// TIA Portal project "OPC_UA_STEP7_CODE_V12" (V14)

(* hardware
DEVICE "SIMATIC 300"  S7-300 station
   slot 0: "UR"  Rail  6ES7 390-1***0-0AA0
   slot 2: "CPU 315-2 PN/DP"  CPU 315-2 PN/DP  6ES7 315-2EH14-0AB0  V3.2
      slot 2: "PROFINET interface_1"  PN-IO
         slot 1: "Port_1"  Port
         slot 2: "Port_2"  Port
   slot 4: "CP 343-1 Advanced-IT_1"  CP 343-1 ADVANCED-IT  6GK7 343-1GX31-0XE0  V3.0
   slot 5: "DI 16/DO 16x24VDC/0.5A"  DI16/DO16 x 24V / 0.5A  6ES7 323-1BL00-0AA0
DEVICE "SIMATIC 400"  S7-400 station
   slot 0: "UR2"  UR2ALU-H  6ES7 400-1JA01-0AA0
   slot 1: "PS 407 10A"  PS 407 10A  6ES7 407-0KA02-0AA0
   slot 3: "CPU 416-3 DP"  CPU 416-3DP  6ES7 416-3XR05-0AB0  V5.1
      slot 1: "DP"  X2
      slot 2: "MPI/DP"  X1
   slot 5: "CP 443-1 Advanced"  CP 443-1 Advanced-IT  6GK7 443-1GX20-0XE0  V2.0
   slot 6: "SM 423 SIM"  DI/DO SIMULATOR  6ES7 423 DI/DO-SIMULATOR
DEVICE "SIMATIC PC Station"  SIMATIC PC station
   slot 0: "PC"  Rail  SIMATIC PC-Station  V1.0
      slot 125: "Stationmanager"  Station_Manager  V6.0.4
   slot 1: "OPC Server"  OPC Server  OPC Server  V14.0.0
   slot 2: "IE General"  IE General  IE_CP  V8.2.0
DEVICE "S71500/ET200MP station_1"  S7-1500 station
   slot 0: "Rail_0"  Rack  6ES7 590-1***0-0AA0
   slot 1: "CPU 1516F-3 PN/DP"  CPU 1516F-3 PN/DP  6ES7 516-3FN00-0AB0  V1.8
      slot 3: "CPU display_1"  6ES7591-1BA00-0AA0
*)

// ===== PLC "CPU 315-2 PN/DP"  CPU 315-2 PN/DP =====

VAR_GLOBAL   // PLC tag table "Default tag table"
   "Tag_1" AT %M100.1 : Bool;
   "Tag_2" AT %M10.6 : Bool;
   "Tag_3" AT %MW302 : Int;
   "Tag_4" AT %MW300 : Int;
   "Tag_5" AT %T1 : Timer;
   "Tag_6" AT %M100.0 : Bool;
END_VAR

VAR_GLOBAL   // PLC tag table "STEP7 classic symbols"
   "CountUP" AT %MB10 : Byte;
END_VAR

DATA_BLOCK "SimulationConfiguration"   // DB10
{ S7_Optimized_Access := 'FALSE' }
VERSION : 0.1
   VAR
      SimulationSpeed : Byte := B#16#10;
      DynamicCharacter : Byte := B#16#20;
      StartASCII : Byte := B#16#20;
      EndASCII : Byte := B#16#7F;
      CurrentStringLength : Byte := B#16#A;
      MaxStringLength : Byte := B#16#A;
      SendDataCountUp : Byte;
      SendDataLength : DWord := DW#16#1000;
   END_VAR
BEGIN
END_DATA_BLOCK

DATA_BLOCK "StaticDataTypes"   // DB50
{ S7_Optimized_Access := 'FALSE' }
VERSION : 0.1
   VAR
      My_Bool : Bool := TRUE;   // Temporary placeholder variable
      My_Integer : Int := -32767;
      My_Byte : Byte := B#16#FF;
      My_Word : Word := W#16#FFFF;
      My_DWord : DWord := DW#16#FFFFFFFF;
      My_DInteger : DInt := L#-2147483647;
      My_Real4 : Real := 1.23456e+0;
      My_Char : Char := 'a';
      My_String10 : String[10] := 'HelloWorld';
      My_DateAndTime : Date_And_Time := DT#10-12-31-12:59:59.123;
   END_VAR
BEGIN
END_DATA_BLOCK

DATA_BLOCK "DynamicDataTypes"   // DB51
{ S7_Optimized_Access := 'FALSE' }
VERSION : 0.1
   VAR
      My_Bool : Bool;   // Temporary placeholder variable
      My_Integer : Int;
      My_Byte : Byte;
      My_Word : Word;
      My_DWord : DWord;
      My_DInteger : DInt;
      My_Real4 : Real;
      My_Char : Char;
      My_String10 : String[10];
      My_DateAndTime : Date_And_Time;
   END_VAR
BEGIN
END_DATA_BLOCK

DATA_BLOCK "InstanceDataBSEND-BRCV"   // DB100
{ S7_Optimized_Access := 'FALSE' }
VERSION : 0.0
// stored: InstanceOfName InvokeBSENDandBRCV
"InvokeBSENDandBRCV"
BEGIN
   BSEND.SD_1 := P#P  0.0 VOID 0;
   BRCV.RD_1 := P#P  0.0 VOID 0;
END_DATA_BLOCK

DATA_BLOCK "SendData"   // DB112
{ S7_Optimized_Access := 'FALSE' }
VERSION : 0.1
   VAR
      SendData : Array[0..4096] of Byte;
   END_VAR
BEGIN
END_DATA_BLOCK

DATA_BLOCK "RcvData"   // DB113
{ S7_Optimized_Access := 'FALSE' }
VERSION : 0.1
   VAR
      RcvData : Array[0..4096] of Byte;
   END_VAR
BEGIN
END_DATA_BLOCK

FUNCTION_BLOCK "InvokeBSENDandBRCV"   // FB100, STL
{ S7_Optimized_Access := 'FALSE' }
VERSION : 0.1
   VAR_INPUT
      INIT_COM : Bool;
   END_VAR
   VAR
      PLC1_COM : Struct
         BSEND_REQ : Bool;
         BSEND_BUSY : Bool;
         BSEND_DONE : Bool;
         BSEND_ERROR : Bool;
         BSEND_COM_START : Bool;   // Pos flank
         BRCV_EN_R : Bool;
         BRCV_BUSY : Bool;
         BRCV_NDR : Bool;
         BRCV_ERROR : Bool;
         BRCV_COM_START : Bool;
         ID : Word;
         BSEND_STATUS : Word;
         BSEND_STAT_SAVE : Word;
         BRCV_STATUS : Word;
         BRCV_STAT_SAVE : Word;
         BSEND_LEN : Word;
         BRCV_LEN : Word;
      END_STRUCT;
      BSEND : BSEND;
      BRCV : BRCV;
   END_VAR
BEGIN

REGION Network 1: Clear BSEND request to start initial communication
         A     #INIT_COM;
         R     #PLC1_COM.BSEND_REQ;
END_REGION

REGION Network 2
   // define the LEN
         A     #INIT_COM;
         JNB   _001;
         L     "SimulationConfiguration".SendDataLength;
         T     #PLC1_COM.BSEND_LEN;
   _001: NOP   0;
END_REGION

REGION Network 3: Invoke BSEND function
         A     #PLC1_COM.BSEND_REQ;
         =     <??.?>;
         BLD   103;
         A     "Tag_1";
         JNB   _002;
         CALL  #BSEND
         ( REQ    := <??.?>,
           R      := ,
           ID     := 16#0001,
           R_ID   := 16#0000_0002,
           DONE   := #PLC1_COM.BSEND_DONE,
           ERROR  := #PLC1_COM.BSEND_ERROR,
           STATUS := #PLC1_COM.BSEND_STATUS,
           SD_1   := P#DB112.DBX0.0 BYTE 4096,
           LEN    := #PLC1_COM.BSEND_LEN
         );
   _002: NOP   0;
END_REGION

REGION Network 4
   // Start BSEND function with the rising edge of the clock marker if the BSEND 
   // function is not busy
   // The REQ input parameter of the BSEND function is triggered with a rising edge 
   // as 
   // long as the BSEND function is not completed!
         AN    "Tag_2";
         S     #PLC1_COM.BSEND_REQ;
         A(;
         O     #PLC1_COM.BSEND_ERROR;
         O     #PLC1_COM.BSEND_DONE;
         );
         R     #PLC1_COM.BSEND_REQ;
         NOP   0;
END_REGION

REGION Network 5: Evaluate STATUS information of the BSEND function
   // If ERROR occured then save STATUS!
         A     #PLC1_COM.BSEND_ERROR;
         JNB   _003;
         L     #PLC1_COM.BSEND_STATUS;
         T     #PLC1_COM.BSEND_STAT_SAVE;
   _003: NOP   0;
END_REGION

REGION Network 6: Invoke BRCV function
         A     "Tag_1";
         =     <??.?>;
         BLD   103;
         A     "Tag_1";
         JNB   _004;
         CALL  #BRCV
         ( EN_R   := <??.?>,
           ID     := 16#0001,
           R_ID   := 16#0000_0001,
           NDR    := #PLC1_COM.BRCV_NDR,
           ERROR  := #PLC1_COM.BRCV_ERROR,
           STATUS := #PLC1_COM.BRCV_STATUS,
           RD_1   := P#DB113.DBX0.0 BYTE 4096,
           LEN    := #PLC1_COM.BRCV_LEN
         );
   _004: NOP   0;
END_REGION

REGION Network 7: Evaluate STATUS information of the BRCV function
   // If ERROR occured then save STATUS!
         A     #PLC1_COM.BRCV_ERROR;
         JNB   _005;
         L     #PLC1_COM.BRCV_STATUS;
         T     #PLC1_COM.BRCV_STAT_SAVE;
   _005: NOP   0;
END_REGION

REGION Network 8: Enable output ENO
         A     "Tag_1";
         SAVE;
END_REGION
END_FUNCTION_BLOCK

FUNCTION "ChangeDateAndTime" : Void   // FC10, STL
{ S7_Optimized_Access := 'FALSE' }
VERSION : 0.1
BEGIN

REGION Network 1
   // Dynamic Date and Time
   //// year
         L     99;
         L     %DB51.DBB34;
         BTI;
         +     1;
         <I;
         JCN   no1;
         L     0;
   no1:  ITB;
         T     %DB51.DBB34;
   //// month
         L     12;
         L     %DB51.DBB35;
         BTI;
         +     1;
         <I;
         JCN   no2;
         L     1;
   no2:  ITB;
         T     %DB51.DBB35;
   //// day
         L     31;
         L     %DB51.DBB36;
         BTI;
         +     1;
         <I;
         JCN   no3;
         L     1;
   no3:  ITB;
         T     %DB51.DBB36;
   //// hour
         L     23;
         L     %DB51.DBB37;
         BTI;
         +     1;
         <I;
         JCN   no4;
         L     0;
   no4:  ITB;
         T     %DB51.DBB37;
   //// minute
         L     59;
         L     %DB51.DBB38;
         BTI;
         +     1;
         <I;
         JCN   no5;
         L     0;
   no5:  ITB;
         T     %DB51.DBB38;
   //// second
         L     59;
         L     %DB51.DBB39;
         BTI;
         +     1;
         <I;
         JCN   no6;
         L     0;
   no6:  ITB;
         T     %DB51.DBB39;
   //// millisecond left part
         L     99;
         L     %DB51.DBB40;
         BTI;
         +     1;
         <I;
         JCN   no7;
         L     0;
   no7:  ITB;
         T     %DB51.DBB40;
   //// millisecond right part
         L     90;
         L     %DB51.DBB41;
         BTI;
         +     10;
         <I;
         JCN   no8;
         L     0;
   no8:  ITB;
         T     %DB51.DBB41;
END_REGION
END_FUNCTION

FUNCTION "ChangeSimpleTypes" : Void   // FC11, STL
{ S7_Optimized_Access := 'FALSE' }
VERSION : 0.1
BEGIN

REGION Network 1: Temporary placeholder variable
   // togle the boolean
         AN    "DynamicDataTypes".My_Bool;
         =     "DynamicDataTypes".My_Bool;
   // increment the byte
         L     "DynamicDataTypes".My_Byte;
         +     1;
         T     "DynamicDataTypes".My_Byte;
   // increment the signed byte
         L     "DynamicDataTypes".My_Char;
         +     1;
         T     "DynamicDataTypes".My_Char;
   // count up by 10
         L     "DynamicDataTypes".My_Word;
         +     10;
         T     "DynamicDataTypes".My_Word;
   // count up by 100
         L     "DynamicDataTypes".My_DWord;
         +     100;
         T     "DynamicDataTypes".My_DWord;
   // count up by 10
         L     "DynamicDataTypes".My_Integer;
         +     10;
         T     "DynamicDataTypes".My_Integer;
   // count up by 100
         L     "DynamicDataTypes".My_DInteger;
         +     100;
         T     "DynamicDataTypes".My_DInteger;
   // count up by 0.1
         L     "DynamicDataTypes".My_Real4;
         L     0.01;
         +R;
         T     "DynamicDataTypes".My_Real4;
END_REGION
END_FUNCTION

FUNCTION "ChangeString" : Void   // FC13, STL
{ S7_Optimized_Access := 'FALSE' }
VERSION : 0.1
BEGIN

REGION Network 1
   // change the content and the length of the string
   // Increment length of dynamic string 10
         L     "SimulationConfiguration".CurrentStringLength;
         L     "SimulationConfiguration".MaxStringLength;
         >=I;
         JC    rst1;

         L     "SimulationConfiguration".CurrentStringLength;
         +     1;
         T     "SimulationConfiguration".CurrentStringLength;
         T     %DB51.DBB23;  //used length of string
         JU    go1;

   rst1: L     1;
         T     "SimulationConfiguration".CurrentStringLength;
         T     %DB51.DBB23;


   // Set new StringChar
   go1:  L     "SimulationConfiguration".DynamicCharacter;
         L     "SimulationConfiguration".EndASCII;  // this is the last letter (ASCII) to use
         >=I;
         JC    rst2;

         L     "SimulationConfiguration".DynamicCharacter;
         +     1;
         T     "SimulationConfiguration".DynamicCharacter;
         JU    go2;

   rst2: L     "SimulationConfiguration".StartASCII;  // this is the first letter (ASCII) to use (32)
         T     "SimulationConfiguration".DynamicCharacter;

   go2:  CALL  FILL
         ( BVAL    := "SimulationConfiguration".DynamicCharacter,
           RET_VAL := "Tag_3",
           BLK     := P#DB51.DBX24.0 BYTE 10
         );
END_REGION
END_FUNCTION

FUNCTION "ChangeSendData" : Void   // FC14, STL
{ S7_Optimized_Access := 'FALSE' }
VERSION : 0.1
BEGIN

REGION Network 1

         L     "SimulationConfiguration".SendDataCountUp;
         L     1;
         +I;
         T     "SimulationConfiguration".SendDataCountUp;
   // take the byte and fill the send buffer
         CALL  FILL
         ( BVAL    := "SimulationConfiguration".SendDataCountUp,
           RET_VAL := "Tag_4",
           BLK     := P#DB112.DBX0.0 BYTE 4096
         );
         NOP   0;
END_REGION
END_FUNCTION

ORGANIZATION_BLOCK "OB1"   // OB1, STL
{ S7_Optimized_Access := 'FALSE' }
VERSION : 0.1
   VAR_TEMP
      TEMP0 : Byte;
      TEMP1 : Byte;
      TEMP2 : Byte;
      TEMP3 : Byte;
      TEMP4 : Byte;
      TEMP5 : Byte;
      TEMP6 : Int;
      TEMP7 : Int;
      TEMP8 : Int;
      TEMP9 : Date_And_Time;
   END_VAR
BEGIN

REGION Network 1: Get a trigger, speed depends on DB10 byte 0
   // check if timer is expired
         AN    "Tag_5";
   // start timer with value global speed variable
         L     "SimulationConfiguration".SimulationSpeed;
         ITB;
         SF    "Tag_5";
         JCN   END;

   // change the values

         CALL  "ChangeDateAndTime";

         CALL  "ChangeSimpleTypes";

         CALL  "ChangeString";

         CALL  "ChangeSendData";

   END:  NOP   0;
END_REGION

REGION Network 2: Activate communication with BSEND/BRCV function
         A     "Tag_6";
         =     <??.?>;
         BLD   103;
         A     "Tag_1";
         JNB   _001;
         CALL  "InvokeBSENDandBRCV", "InstanceDataBSEND-BRCV"
         ( INIT_COM := <??.?>
         );

   _001: A     BR;
         R     "Tag_6";
END_REGION
END_ORGANIZATION_BLOCK

ORGANIZATION_BLOCK "OB100"   // OB100, STL
TITLE = "Complete Restart"
{ S7_Optimized_Access := 'FALSE' }
VERSION : 0.1
   VAR_TEMP
      OB100_EV_CLASS : Byte;   // 16#13, Event class 1, Entering event state, Event logged in diagnostic buffer
      OB100_STRTUP : Byte;   // 16#81/82/83/84 Method of startup
      OB100_PRIORITY : Byte;   // Priority of OB Execution
      OB100_OB_NUMBR : Byte;   // 100 (Organization block 100, OB100)
      OB100_RESERVED_1 : Byte;   // Reserved for system
      OB100_RESERVED_2 : Byte;   // Reserved for system
      OB100_STOP : Word;   // Event that caused CPU to stop (16#4xxx)
      OB100_STRT_INFO : DWord;   // Information on how system started
      OB100_DATE_TIME : Date_And_Time;   // Date and time OB100 started
   END_VAR
BEGIN

REGION Network 1: Enable communication function blocks

         AN    "Tag_6";
         S     "Tag_6";
END_REGION

REGION Network 2: Force restart of communication block
         AN    "Tag_1";
         S     "Tag_1";
END_REGION
END_ORGANIZATION_BLOCK

// ===== PLC "CPU 416-3 DP"  CPU 416-3DP =====

VAR_GLOBAL   // PLC tag table "Default tag table"
   "Tag_1" AT %M100.1 : Bool;
   "Tag_2" AT %M10.6 : Bool;
   "Tag_3" AT %MW302 : Int;
   "Tag_4" AT %MW300 : Int;
   "Tag_5" AT %T1 : Timer;
   "Tag_6" AT %M100.0 : Bool;
END_VAR

VAR_GLOBAL   // PLC tag table "STEP7 classic symbols"
   "CountUP" AT %MB10 : Byte;
END_VAR

DATA_BLOCK "SimulationConfiguration"   // DB10
{ S7_Optimized_Access := 'FALSE' }
VERSION : 0.1
   VAR
      SimulationSpeed : Byte := B#16#10;
      DynamicCharacter : Byte := B#16#20;
      StartASCII : Byte := B#16#20;
      EndASCII : Byte := B#16#7F;
      CurrentStringLength : Byte := B#16#A;
      MaxStringLength : Byte := B#16#A;
      SendDataCountUp : Byte;
      SendDataLength : DWord := DW#16#1000;
   END_VAR
BEGIN
END_DATA_BLOCK

DATA_BLOCK "StaticDataTypes"   // DB50
{ S7_Optimized_Access := 'FALSE' }
VERSION : 0.1
   VAR
      My_Bool : Bool := TRUE;   // Temporary placeholder variable
      My_Integer : Int := -32767;
      My_Byte : Byte := B#16#FF;
      My_Word : Word := W#16#FFFF;
      My_DWord : DWord := DW#16#FFFFFFFF;
      My_DInteger : DInt := L#-2147483647;
      My_Real4 : Real := 1.23456e+0;
      My_Char : Char := 'a';
      My_String10 : String[10] := 'HelloWorld';
      My_DateAndTime : Date_And_Time := DT#10-12-31-12:59:59.123;
   END_VAR
BEGIN
END_DATA_BLOCK

DATA_BLOCK "DynamicDataTypes"   // DB51
{ S7_Optimized_Access := 'FALSE' }
VERSION : 0.1
   VAR
      My_Bool : Bool;   // Temporary placeholder variable
      My_Integer : Int;
      My_Byte : Byte;
      My_Word : Word;
      My_DWord : DWord;
      My_DInteger : DInt;
      My_Real4 : Real;
      My_Char : Char;
      My_String10 : String[10];
      My_DateAndTime : Date_And_Time;
   END_VAR
BEGIN
END_DATA_BLOCK

DATA_BLOCK "InstanceDataBSEND-BRCV"   // DB100
{ S7_Optimized_Access := 'FALSE' }
VERSION : 0.0
// stored: InstanceOfName InvokeBSENDandBRCV
"InvokeBSENDandBRCV"
BEGIN
END_DATA_BLOCK

DATA_BLOCK "SendData"   // DB112
{ S7_Optimized_Access := 'FALSE' }
VERSION : 0.1
   VAR
      SendData : Array[0..4096] of Byte;
   END_VAR
BEGIN
END_DATA_BLOCK

DATA_BLOCK "RcvData"   // DB113
{ S7_Optimized_Access := 'FALSE' }
VERSION : 0.1
   VAR
      RcvData : Array[0..4096] of Byte;
   END_VAR
BEGIN
END_DATA_BLOCK

FUNCTION_BLOCK "InvokeBSENDandBRCV"   // FB100, STL
{ S7_Optimized_Access := 'FALSE' }
VERSION : 0.1
   VAR_INPUT
      INIT_COM : Bool;
   END_VAR
   VAR
      PLC1_COM : Struct
         BSEND_REQ : Bool;
         BSEND_BUSY : Bool;
         BSEND_DONE : Bool;
         BSEND_ERROR : Bool;
         BSEND_COM_START : Bool;   // Pos flank
         BRCV_EN_R : Bool;
         BRCV_BUSY : Bool;
         BRCV_NDR : Bool;
         BRCV_ERROR : Bool;
         BRCV_COM_START : Bool;
         ID : Word;
         BSEND_STATUS : Word;
         BSEND_STAT_SAVE : Word;
         BRCV_STATUS : Word;
         BRCV_STAT_SAVE : Word;
         BSEND_LEN : Word;
         BRCV_LEN : Word;
      END_STRUCT;
   END_VAR
BEGIN

REGION Network 1: Clear BSEND request to start initial communication
         A     #INIT_COM;
         R     #PLC1_COM.BSEND_REQ;
END_REGION

REGION Network 2
   // define the LEN
         A     #INIT_COM;
         JNB   _001;
         L     "SimulationConfiguration".SendDataLength;
         T     #PLC1_COM.BSEND_LEN;
   _001: NOP   0;
END_REGION

REGION Network 3: Invoke BSEND function
         A     #PLC1_COM.BSEND_REQ;
         =     <??.?>;
         BLD   103;
         A     "Tag_1";
         JNB   _002;
         CALL  BSEND, "DB12"
         ( REQ    := <??.?>,
           R      := ,
           ID     := 16#0001,
           R_ID   := 16#0000_0001,
           DONE   := #PLC1_COM.BSEND_DONE,
           ERROR  := #PLC1_COM.BSEND_ERROR,
           STATUS := #PLC1_COM.BSEND_STATUS,
           SD_1   := P#DB112.DBX0.0 BYTE 4096,
           LEN    := #PLC1_COM.BSEND_LEN
         );
   _002: NOP   0;
END_REGION

REGION Network 4
   // Start BSEND function with the rising edge of the clock marker if the BSEND 
   // function is not busy
   // The REQ input parameter of the BSEND function is triggered with a rising edge 
   // as 
   // long as the BSEND function is not completed!
         AN    "Tag_2";
         S     #PLC1_COM.BSEND_REQ;
         A(;
         O     #PLC1_COM.BSEND_ERROR;
         O     #PLC1_COM.BSEND_DONE;
         );
         R     #PLC1_COM.BSEND_REQ;
         NOP   0;
END_REGION

REGION Network 5: Evaluate STATUS information of the BSEND function
   // If ERROR occured then save STATUS!
         A     #PLC1_COM.BSEND_ERROR;
         JNB   _003;
         L     #PLC1_COM.BSEND_STATUS;
         T     #PLC1_COM.BSEND_STAT_SAVE;
   _003: NOP   0;
END_REGION

REGION Network 6: Invoke BRCV function
         A     "Tag_1";
         =     <??.?>;
         BLD   103;
         A     "Tag_1";
         JNB   _004;
         CALL  BRCV, "DB13"
         ( EN_R   := <??.?>,
           ID     := 16#0001,
           R_ID   := 16#0000_0001,
           NDR    := #PLC1_COM.BRCV_NDR,
           ERROR  := #PLC1_COM.BRCV_ERROR,
           STATUS := #PLC1_COM.BRCV_STATUS,
           RD_1   := P#DB113.DBX0.0 BYTE 4096,
           LEN    := #PLC1_COM.BRCV_LEN
         );
   _004: NOP   0;
END_REGION

REGION Network 7: Evaluate STATUS information of the BRCV function
   // If ERROR occured then save STATUS!
         A     #PLC1_COM.BRCV_ERROR;
         JNB   _005;
         L     #PLC1_COM.BRCV_STATUS;
         T     #PLC1_COM.BRCV_STAT_SAVE;
   _005: NOP   0;
END_REGION

REGION Network 8: Enable output ENO
         A     "Tag_1";
         SAVE;
END_REGION
END_FUNCTION_BLOCK

FUNCTION "ChangeDateAndTime" : Void   // FC10, STL
{ S7_Optimized_Access := 'FALSE' }
VERSION : 0.1
BEGIN

REGION Network 1
   // Dynamic Date and Time
   //// year
         L     99;
         L     %DB51.DBB34;
         BTI;
         +     1;
         <I;
         JCN   no1;
         L     0;
   no1:  ITB;
         T     %DB51.DBB34;
   //// month
         L     12;
         L     %DB51.DBB35;
         BTI;
         +     1;
         <I;
         JCN   no2;
         L     1;
   no2:  ITB;
         T     %DB51.DBB35;
   //// day
         L     31;
         L     %DB51.DBB36;
         BTI;
         +     1;
         <I;
         JCN   no3;
         L     1;
   no3:  ITB;
         T     %DB51.DBB36;
   //// hour
         L     23;
         L     %DB51.DBB37;
         BTI;
         +     1;
         <I;
         JCN   no4;
         L     0;
   no4:  ITB;
         T     %DB51.DBB37;
   //// minute
         L     59;
         L     %DB51.DBB38;
         BTI;
         +     1;
         <I;
         JCN   no5;
         L     0;
   no5:  ITB;
         T     %DB51.DBB38;
   //// second
         L     59;
         L     %DB51.DBB39;
         BTI;
         +     1;
         <I;
         JCN   no6;
         L     0;
   no6:  ITB;
         T     %DB51.DBB39;
   //// millisecond left part
         L     99;
         L     %DB51.DBB40;
         BTI;
         +     1;
         <I;
         JCN   no7;
         L     0;
   no7:  ITB;
         T     %DB51.DBB40;
   //// millisecond right part
         L     90;
         L     %DB51.DBB41;
         BTI;
         +     10;
         <I;
         JCN   no8;
         L     0;
   no8:  ITB;
         T     %DB51.DBB41;
END_REGION
END_FUNCTION

FUNCTION "ChangeSimpleTypes" : Void   // FC11, STL
{ S7_Optimized_Access := 'FALSE' }
VERSION : 0.1
BEGIN

REGION Network 1: Temporary placeholder variable
   // togle the boolean
         AN    "DynamicDataTypes".My_Bool;
         =     "DynamicDataTypes".My_Bool;
   // increment the byte
         L     "DynamicDataTypes".My_Byte;
         +     1;
         T     "DynamicDataTypes".My_Byte;
   // increment the signed byte
         L     "DynamicDataTypes".My_Char;
         +     1;
         T     "DynamicDataTypes".My_Char;
   // count up by 10
         L     "DynamicDataTypes".My_Word;
         +     10;
         T     "DynamicDataTypes".My_Word;
   // count up by 100
         L     "DynamicDataTypes".My_DWord;
         +     100;
         T     "DynamicDataTypes".My_DWord;
   // count up by 10
         L     "DynamicDataTypes".My_Integer;
         +     10;
         T     "DynamicDataTypes".My_Integer;
   // count up by 100
         L     "DynamicDataTypes".My_DInteger;
         +     100;
         T     "DynamicDataTypes".My_DInteger;
   // count up by 0.1
         L     "DynamicDataTypes".My_Real4;
         L     0.01;
         +R;
         T     "DynamicDataTypes".My_Real4;
END_REGION
END_FUNCTION

FUNCTION "ChangeString" : Void   // FC13, STL
{ S7_Optimized_Access := 'FALSE' }
VERSION : 0.1
BEGIN

REGION Network 1
   // change the content and the length of the string
   // Increment length of dynamic string 10
         L     "SimulationConfiguration".CurrentStringLength;
         L     "SimulationConfiguration".MaxStringLength;
         >=I;
         JC    rst1;

         L     "SimulationConfiguration".CurrentStringLength;
         +     1;
         T     "SimulationConfiguration".CurrentStringLength;
         T     %DB51.DBB23;  //used length of string
         JU    go1;

   rst1: L     1;
         T     "SimulationConfiguration".CurrentStringLength;
         T     %DB51.DBB23;


   // Set new StringChar
   go1:  L     "SimulationConfiguration".DynamicCharacter;
         L     "SimulationConfiguration".EndASCII;  // this is the last letter (ASCII) to use
         >=I;
         JC    rst2;

         L     "SimulationConfiguration".DynamicCharacter;
         +     1;
         T     "SimulationConfiguration".DynamicCharacter;
         JU    go2;

   rst2: L     "SimulationConfiguration".StartASCII;  // this is the first letter (ASCII) to use (32)
         T     "SimulationConfiguration".DynamicCharacter;

   go2:  CALL  FILL
         ( BVAL    := "SimulationConfiguration".DynamicCharacter,
           RET_VAL := "Tag_3",
           BLK     := P#DB51.DBX24.0 BYTE 10
         );
END_REGION
END_FUNCTION

FUNCTION "ChangeSendData" : Void   // FC14, STL
{ S7_Optimized_Access := 'FALSE' }
VERSION : 0.1
BEGIN

REGION Network 1
         L     "SimulationConfiguration".SendDataCountUp;
         L     1;
         +I;
         T     "SimulationConfiguration".SendDataCountUp;
   // take the byte and fill the send buffer
         CALL  FILL
         ( BVAL    := "SimulationConfiguration".SendDataCountUp,
           RET_VAL := "Tag_4",
           BLK     := P#DB112.DBX0.0 BYTE 4096
         );
         NOP   0;
END_REGION
END_FUNCTION

ORGANIZATION_BLOCK "OB1"   // OB1, STL
{ S7_Optimized_Access := 'FALSE' }
VERSION : 0.1
   VAR_TEMP
      TEMP0 : Byte;
      TEMP1 : Byte;
      TEMP2 : Byte;
      TEMP3 : Byte;
      TEMP4 : Byte;
      TEMP5 : Byte;
      TEMP6 : Int;
      TEMP7 : Int;
      TEMP8 : Int;
      TEMP9 : Date_And_Time;
   END_VAR
BEGIN

REGION Network 1: Get a trigger, speed depends on DB10 byte 0
   // check if timer is expired
         AN    "Tag_5";
   // start timer with value global speed variable
         L     "SimulationConfiguration".SimulationSpeed;
         ITB;
         SF    "Tag_5";
         JCN   END;

   // change the values

         CALL  "ChangeDateAndTime";

         CALL  "ChangeSimpleTypes";

         CALL  "ChangeString";

         CALL  "ChangeSendData";

   END:  NOP   0;
END_REGION

REGION Network 2: Activate communication with BSEND/BRCV function
         A     "Tag_6";
         =     <??.?>;
         BLD   103;
         A     "Tag_1";
         JNB   _001;
         CALL  "InvokeBSENDandBRCV", "InstanceDataBSEND-BRCV"
         ( INIT_COM := <??.?>
         );

   _001: A     BR;
         R     "Tag_6";
END_REGION
END_ORGANIZATION_BLOCK

ORGANIZATION_BLOCK "OB100"   // OB100, STL
TITLE = "Complete Restart"
{ S7_Optimized_Access := 'FALSE' }
VERSION : 0.1
   VAR_TEMP
      OB100_EV_CLASS : Byte;   // 16#13, Event class 1, Entering event state, Event logged in diagnostic buffer
      OB100_STRTUP : Byte;   // 16#81/82/83/84 Method of startup
      OB100_PRIORITY : Byte;   // Priority of OB Execution
      OB100_OB_NUMBR : Byte;   // 100 (Organization block 100, OB100)
      OB100_RESERVED_1 : Byte;   // Reserved for system
      OB100_RESERVED_2 : Byte;   // Reserved for system
      OB100_STOP : Word;   // Event that caused CPU to stop (16#4xxx)
      OB100_STRT_INFO : DWord;   // Information on how system started
      OB100_DATE_TIME : Date_And_Time;   // Date and time OB100 started
   END_VAR
BEGIN

REGION Network 1: Enable communication function blocks

         AN    "Tag_6";
         S     "Tag_6";
END_REGION

REGION Network 2: Force restart of communication block
         AN    "Tag_1";
         S     "Tag_1";
END_REGION
END_ORGANIZATION_BLOCK

// ===== PLC "CPU 1516F-3 PN/DP"  CPU 1516F-3 PN/DP =====

DATA_BLOCK "StaticDataTypesOpt"   // DB1
{ S7_Optimized_Access := 'TRUE' }
VERSION : 0.1
   VAR
      My_Bool : Bool := TRUE;   // Temporary placeholder variable
      My_Integer : Int := -32767;
      My_Byte : Byte := B#16#FF;
      My_Word : Word := W#16#FFFF;
      My_DWord : DWord := DW#16#FFFFFFFF;
      My_DInteger : DInt := L#-2147483647;
      My_Real4 : Real := 1.23456;
      My_Char : Char := 'a';
      My_String10 : String[10] := 'HelloWorld';
      My_DateAndTime : Date_And_Time := DT#10-12-31-12:59:59.123;
   END_VAR
BEGIN
END_DATA_BLOCK

DATA_BLOCK "StaticDataTypesNonOpt"   // DB2
{ S7_Optimized_Access := 'FALSE' }
VERSION : 0.1
   VAR
      My_Bool : Bool := TRUE;   // Temporary placeholder variable
      My_Integer : Int := -32767;
      My_Byte : Byte := B#16#FF;
      My_Word : Word := W#16#FFFF;
      My_DWord : DWord := DW#16#FFFFFFFF;
      My_DInteger : DInt := L#-2147483647;
      My_Real4 : Real := 1.23456;
      My_Char : Char := 'a';
      My_String10 : String[10] := 'HelloWorld';
      My_DateAndTime : Date_And_Time := DT#10-12-31-12:59:59.123;
   END_VAR
BEGIN
END_DATA_BLOCK

ORGANIZATION_BLOCK "Main"   // OB1, LAD, ProgramCycle
TITLE = "Main Program Sweep (Cycle)"
{ S7_Optimized_Access := 'TRUE' }
VERSION : 0.1
   VAR_INPUT
      Initial_Call : Bool;   // Initial call of this OB
      Remanence : Bool;   // =True, if remanent data are available
   END_VAR
BEGIN
END_ORGANIZATION_BLOCK